    PROC writeCursive(string sText)
        VAR num i;
        VAR string sChar;
        FOR i FROM 1 TO StrLen(sText) DO
            sChar := StrPart(sText,i,1);
            TEST sChar
                CASE "a":
                    char_a;
                CASE "b":
                    char_b;
                CASE "c":
                    char_c;
                CASE "d":
                    char_d;
                CASE "e":
                    char_e;
                CASE "f":
                    char_f;
                CASE "g":
                    char_g;
                CASE "h":
                    char_h;
                CASE "i":
                    char_i;
                CASE "j":
                    char_j;
                CASE "k":
                    char_k;
                CASE "l":
                    char_l;
                CASE "m":
                    char_m;
                CASE "n":
                    char_n;
                CASE "o":
                    char_o;
                CASE "p":
                    char_p;
                CASE "q":
                    char_q;
                CASE "r":
                    char_r;
                CASE "s":
                    char_s;
                CASE "t":
                    char_t;
                CASE "u":
                    char_u;
                CASE "v":
                    char_v;
                CASE "w":
                    char_w;
                CASE "x":
                    char_x;
                CASE "y":
                    char_y;
                CASE "z":
                    char_z;
                CASE "A":
                    char_upperA;
                CASE "B":
                    char_upperB;
                CASE "C":
                    char_upperC;
                CASE "D":
                    char_upperD;
                CASE "E":
                    char_upperE;
                CASE "F":
                    char_upperF;
                CASE "G":
                    char_upperG;
                CASE "H":
                    char_upperH;
                CASE "I":
                    char_upperI;
                CASE "J":
                    char_upperJ;
                CASE "K":
                    char_upperK;
                CASE "L":
                    char_upperL;
                CASE "M":
                    char_upperM;
                CASE "N":
                    char_upperN;
                CASE "O":
                    char_upperO;
                CASE "P":
                    char_upperP;
                CASE "Q":
                    char_upperQ;
                CASE "R":
                    char_upperR;
                CASE "S":
                    char_upperS;
                CASE "T":
                    char_upperT;
                CASE "U":
                    char_upperU;
                CASE "V":
                    char_upperV;
                CASE "W":
                    char_upperW;
                CASE "X":
                    char_upperX;
                CASE "Y":
                    char_upperY;
                CASE "Z":
                    char_upperZ;
                CASE "0":
                    char_0;
                CASE "1":
                    char_1;
                CASE "2":
                    char_2;
                CASE "3":
                    char_3;
                CASE "4":
                    char_4;
                CASE "5":
                    char_5;
                CASE "6":
                    char_6;
                CASE "7":
                    char_7;
                CASE "8":
                    char_8;
                CASE "9":
                    char_9;
                CASE "!":
                    char_exclamation;
                CASE "@":
                    char_at;
                CASE "#":
                    char_hash;
                CASE "$":
                    char_dollar;
                CASE "%":
                    char_percent;
                CASE "^":
                    char_caret;
                CASE "&":
                    char_ampersand;
                CASE "*":
                    char_asterisk;
                CASE "(":
                    char_leftparenthesis;
                CASE ")":
                    char_rightparenthesis;
                CASE "+":
                    char_plus;
                CASE "=":
                    char_equals;
                CASE "[":
                    char_leftbracket;
                CASE "]":
                    char_rightbracket;
                CASE "{":
                    char_leftbrace;
                CASE "}":
                    char_rightbrace;
                CASE "|":
                    char_pipe;
                CASE "<":
                    char_lessthan;
                CASE ">":
                    char_greaterthan;
                CASE "?":
                    char_question;
                CASE "_":
                    char_underscore;
                CASE "-":
                    char_minus;
                CASE "~":
                    char_tilde;
                CASE ".":
                    char_period;
                CASE ",":
                    char_comma;
                CASE ";":
                    char_semicolon;
                CASE ":":
                    char_colon;
                CASE " ":
                    ! Space - move right without drawing
                    wWobj.oframe.trans.x := wWobj.oframe.trans.x + 15;
                DEFAULT:
                    TPWrite "Character not supported: " + sChar;
            ENDTEST
        ENDFOR
    ENDPROC
ENDMODULE

--- Controller Data/IRB1200_5_90/SYSPAR/EIO.cfg ---
EIO:CFG_1.0:7:0::
#
VIRTUAL_NETWORK:

      -Name "Virtual" -Label "Virtual Device Network"
#
EIO_SIGNAL:

      -Name "IIO_di1" -SignalType "DI" -Device "IntegratedIOInternalDevice"\
      -DeviceMap "0"

      -Name "IIO_di2" -SignalType "DI" -Device "IntegratedIOInternalDevice"\
      -DeviceMap "1"

      -Name "IIO_di3" -SignalType "DI" -Device "IntegratedIOInternalDevice"\
      -DeviceMap "2"

      -Name "IIO_di4" -SignalType "DI" -Device "IntegratedIOInternalDevice"\
      -DeviceMap "3"

      -Name "IIO_di5" -SignalType "DI" -Device "IntegratedIOInternalDevice"\
      -DeviceMap "4"

      -Name "IIO_di6" -SignalType "DI" -Device "IntegratedIOInternalDevice"\
      -DeviceMap "5"

      -Name "IIO_di7" -SignalType "DI" -Device "IntegratedIOInternalDevice"\
      -DeviceMap "6"

      -Name "IIO_di8" -SignalType "DI" -Device "IntegratedIOInternalDevice"\
      -DeviceMap "7"

      -Name "IIO_di9" -SignalType "DI" -Device "IntegratedIOInternalDevice"\
      -DeviceMap "8"

      -Name "IIO_di10" -SignalType "DI" -Device "IntegratedIOInternalDevice"\
      -DeviceMap "9"

      -Name "IIO_di11" -SignalType "DI" -Device "IntegratedIOInternalDevice"\
      -DeviceMap "10"

      -Name "IIO_di12" -SignalType "DI" -Device "IntegratedIOInternalDevice"\
      -DeviceMap "11"

      -Name "IIO_di13" -SignalType "DI" -Device "IntegratedIOInternalDevice"\
      -DeviceMap "12"

      -Name "IIO_di14" -SignalType "DI" -Device "IntegratedIOInternalDevice"\
      -DeviceMap "13"

      -Name "IIO_di15" -SignalType "DI" -Device "IntegratedIOInternalDevice"\
      -DeviceMap "14"

      -Name "IIO_di16" -SignalType "DI" -Device "IntegratedIOInternalDevice"\
      -DeviceMap "15"

      -Name "IIO_do1" -SignalType "DO" -Device "IntegratedIOInternalDevice"\
      -DeviceMap "0"

      -Name "IIO_do2" -SignalType "DO" -Device "IntegratedIOInternalDevice"\
      -DeviceMap "1"

      -Name "IIO_do3" -SignalType "DO" -Device "IntegratedIOInternalDevice"\
      -DeviceMap "2"

      -Name "IIO_do4" -SignalType "DO" -Device "IntegratedIOInternalDevice"\
      -DeviceMap "3"

      -Name "IIO_do5" -SignalType "DO" -Device "IntegratedIOInternalDevice"\
      -DeviceMap "4"

      -Name "IIO_do6" -SignalType "DO" -Device "IntegratedIOInternalDevice"\
      -DeviceMap "5"

      -Name "IIO_do7" -SignalType "DO" -Device "IntegratedIOInternalDevice"\
      -DeviceMap "6"

      -Name "IIO_do8" -SignalType "DO" -Device "IntegratedIOInternalDevice"\
      -DeviceMap "7"

      -Name "IIO_gi" -SignalType "GI" -Device "integratedIOInternalDevice"\
      -DeviceMap "0-15"

      -Name "IIO_go" -SignalType "GO" -Device "integratedIOInternalDevice"\
      -DeviceMap "0-7"

      -Name "do_pen" -SignalType "DO" -Access "All"

#CTRL_SIGNATURE:UpI3rsGsdjPUEdBBGvNwuUTXFijTMgTtD42mLhnlGZgDW7Y00ZW5+aDJae9I93WBev467PSv26CaKbAkbr5rXw==

--- Controller Data/IRB1200_5_90/SYSPAR/PROC.cfg ---
PROC:CFG_1.0:7:0::

#CTRL_SIGNATURE:EanoTt332vqhZPmKvdzBrByTheeXv3GTX9o65SYsnrJ+DJbQQ2h+v49xbjzxd2tjmmEe4Rias40o22ORGzDJ/w==
